VAR_GLOBAL
	    {attribute 'hide'}
		fbLogger:			FB_Logger;
END_VAR

(* stored: Version 1.1.0.1
   GVL GLV: Id {470c2b31-7e29-075f-0fd9-081ad8199996} *)
